// TIA Portal V15.1 export
// export: Created 2020-06-12T07:35:52.4755859Z, ExportSetting None, DisplayName Totally Integrated Automation Portal, DisplayVersion V15.1, DisplayName TIA Portal Openness, DisplayVersion V15.1, DisplayName STEP 7 Professional, DisplayVersion V15.1, DisplayName STEP 7 Safety, DisplayVersion V15.1, DisplayName WinCC Advanced, DisplayVersion V15.1
FUNCTION "MELT_Meas" : Void   // FC123, FBD
TITLE = Melt process measurements
{ S7_Optimized_Access := 'TRUE' }
// stored: SetENOAutomatically False
   VAR_TEMP
      trigger_ST : Bool;
      trigger_MT : Bool;
      trigger_HT : Bool;
      tTmpU : Real;
      tPower_set : Real;
      tReset_tara : Bool;
      tLimit : Bool;
      tAct_wt : Real;
      tWt_pres : Real;
      tWt_corr : Real;
      tWeight_av : Real;
      tMr_pres : Real;
      tPrs_corr : Real;
      tReset : Bool;
      tFactor : Real;
      tOperator_buttons_ok : Bool;
      tHt_ingot : Bool;
      tIngot_type : DInt;
      tConst_lim2_del_off : Bool;
      txxx : Bool;
      tSlag_molten : Bool;
      tClk_mr : Bool;
      tClk_sw : Bool;
      tCycle_mr : Time;
      tCycle_sw : Time;
      tWeight_av_1 : Real;
      tKWt : Real;
      par500 : Bool;
      par800 : Bool;
      par1050 : Bool;
      par1250 : Bool;
      tTot_ST : Real;
      tTot_time : Real;
      tTmp_time : Time;
      tT_ht : Time;
      tMeltrate1 : Real;
      tMeltrate2 : Real;
      tResMean : Real;
      tResStdDev : Real;
      tSync1 : Bool;
      tSync2 : Bool;
      tCTime1 : Time;
      tCTime2 : Time;
      tMRerr : Real;
      tSWerr : Real;
   END_VAR
BEGIN

REGION Network 1: Actual Power, kW
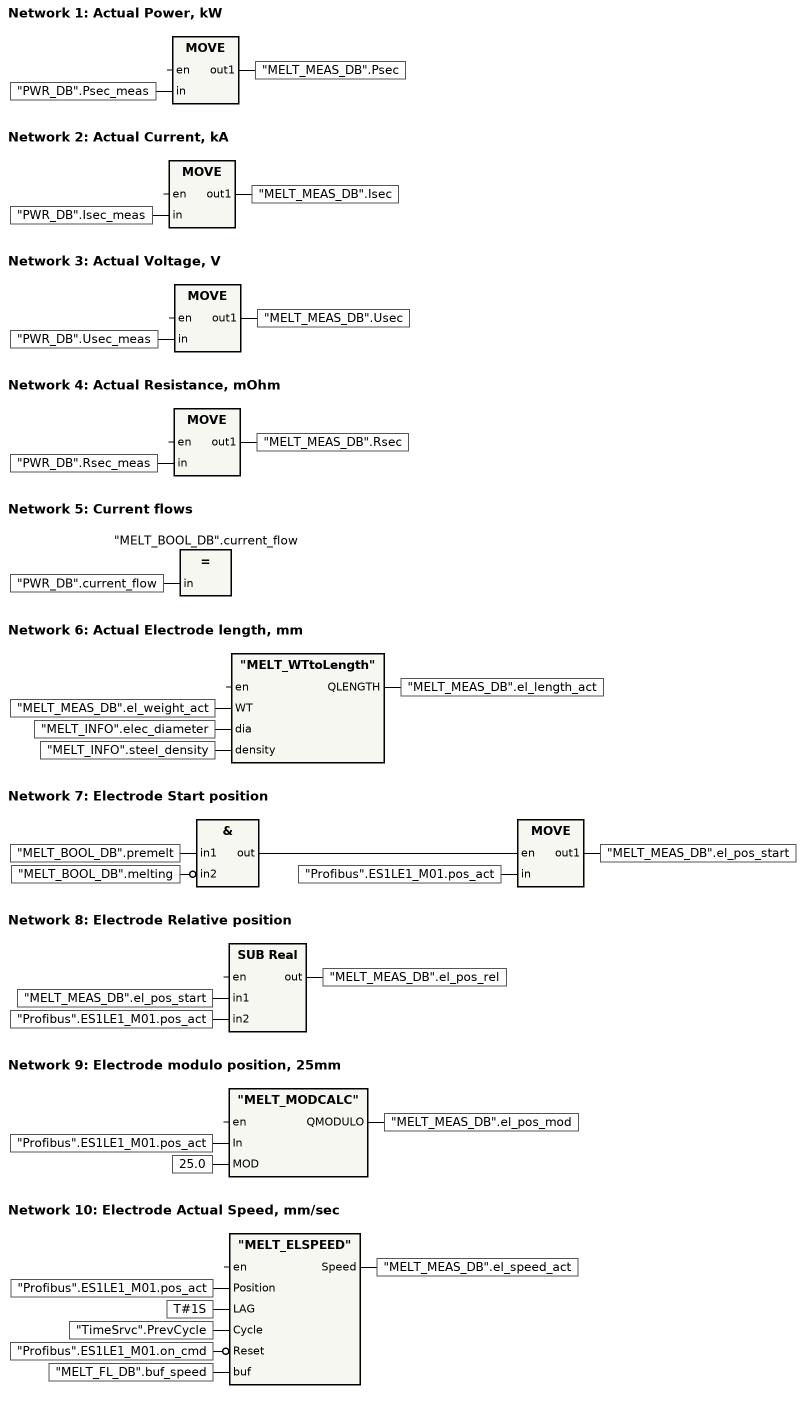
   "MELT_MEAS_DB".Psec := "PWR_DB".Psec_meas;
END_REGION

REGION Network 2: Actual Current, kA
   "MELT_MEAS_DB".Isec := "PWR_DB".Isec_meas;
END_REGION

REGION Network 3: Actual Voltage, V
   "MELT_MEAS_DB".Usec := "PWR_DB".Usec_meas;
END_REGION

REGION Network 4: Actual Resistance, mOhm
   "MELT_MEAS_DB".Rsec := "PWR_DB".Rsec_meas;
END_REGION

REGION Network 5: Current flows
   "MELT_BOOL_DB".current_flow := "PWR_DB".current_flow;
END_REGION

REGION Network 6: Actual Electrode length, mm
   "MELT_WTtoLength"(WT := "MELT_MEAS_DB".el_weight_act,
                     dia := "MELT_INFO".elec_diameter,
                     density := "MELT_INFO".steel_density,
                     QLENGTH => "MELT_MEAS_DB".el_length_act);
END_REGION

REGION Network 7: Electrode Start position
   IF "MELT_BOOL_DB".premelt AND NOT "MELT_BOOL_DB".melting THEN
       "MELT_MEAS_DB".el_pos_start := "Profibus".ES1LE1_M01.pos_act;
   END_IF;
END_REGION

REGION Network 8: Electrode Relative position
   "MELT_MEAS_DB".el_pos_rel := "MELT_MEAS_DB".el_pos_start - "Profibus".ES1LE1_M01.pos_act;
END_REGION

REGION Network 9: Electrode modulo position, 25mm
   "MELT_MODCALC"(In := "Profibus".ES1LE1_M01.pos_act, "MOD" := 25.0, QMODULO => "MELT_MEAS_DB".el_pos_mod);
END_REGION

REGION Network 10: Electrode Actual Speed, mm/sec
   "MELT_ELSPEED"(Position := "Profibus".ES1LE1_M01.pos_act,
                  LAG := T#1S,
                  Cycle := "TimeSrvc".PrevCycle,
                  Reset := NOT "Profibus".ES1LE1_M01.on_cmd,
                  buf := "MELT_FL_DB".buf_speed,
                  Speed => "MELT_MEAS_DB".el_speed_act);
END_REGION

REGION Network 11: Actual Ingot weight
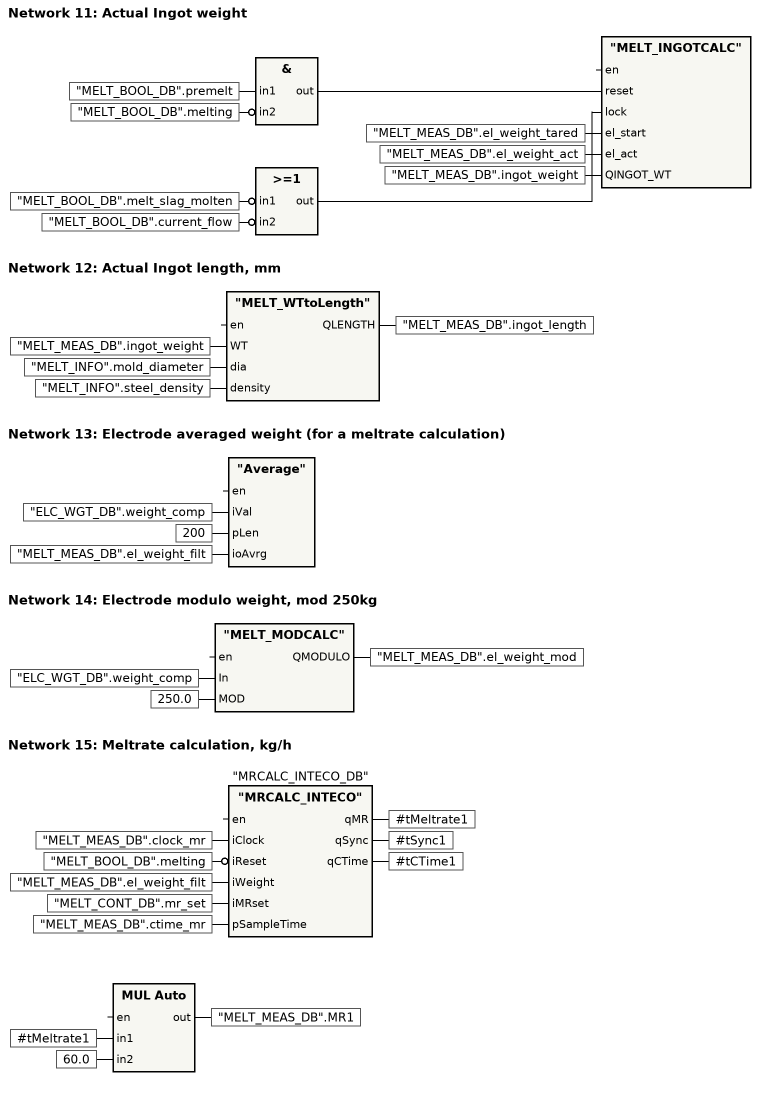
   "MELT_INGOTCALC"(reset := "MELT_BOOL_DB".premelt AND NOT "MELT_BOOL_DB".melting,
                    lock := NOT "MELT_BOOL_DB".melt_slag_molten OR NOT "MELT_BOOL_DB".current_flow,
                    el_start := "MELT_MEAS_DB".el_weight_tared,
                    el_act := "MELT_MEAS_DB".el_weight_act,
                    QINGOT_WT := "MELT_MEAS_DB".ingot_weight);
END_REGION

REGION Network 12: Actual Ingot length, mm
   "MELT_WTtoLength"(WT := "MELT_MEAS_DB".ingot_weight,
                     dia := "MELT_INFO".mold_diameter,
                     density := "MELT_INFO".steel_density,
                     QLENGTH => "MELT_MEAS_DB".ingot_length);
END_REGION

REGION Network 13: Electrode averaged weight (for a meltrate calculation)
   "Average"(iVal := "ELC_WGT_DB".weight_comp, pLen := 200, ioAvrg := "MELT_MEAS_DB".el_weight_filt);
END_REGION

REGION Network 14: Electrode modulo weight, mod 250kg
   "MELT_MODCALC"(In := "ELC_WGT_DB".weight_comp, "MOD" := 250.0, QMODULO => "MELT_MEAS_DB".el_weight_mod);
END_REGION

REGION Network 15: Meltrate calculation, kg/h
   "MRCALC_INTECO_DB"(iClock := "MELT_MEAS_DB".clock_mr,   // "MRCALC_INTECO"
                      iReset := NOT "MELT_BOOL_DB".melting,
                      iWeight := "MELT_MEAS_DB".el_weight_filt,
                      iMRset := "MELT_CONT_DB".mr_set,
                      pSampleTime := "MELT_MEAS_DB".ctime_mr,
                      qMR => #tMeltrate1,
                      qSync => #tSync1,
                      qCTime => #tCTime1);
   "MELT_MEAS_DB".MR1 := #tMeltrate1 * 60.0;
END_REGION

REGION Network 16: Meltrate calculation, kg/h (new)
   // from Boehler
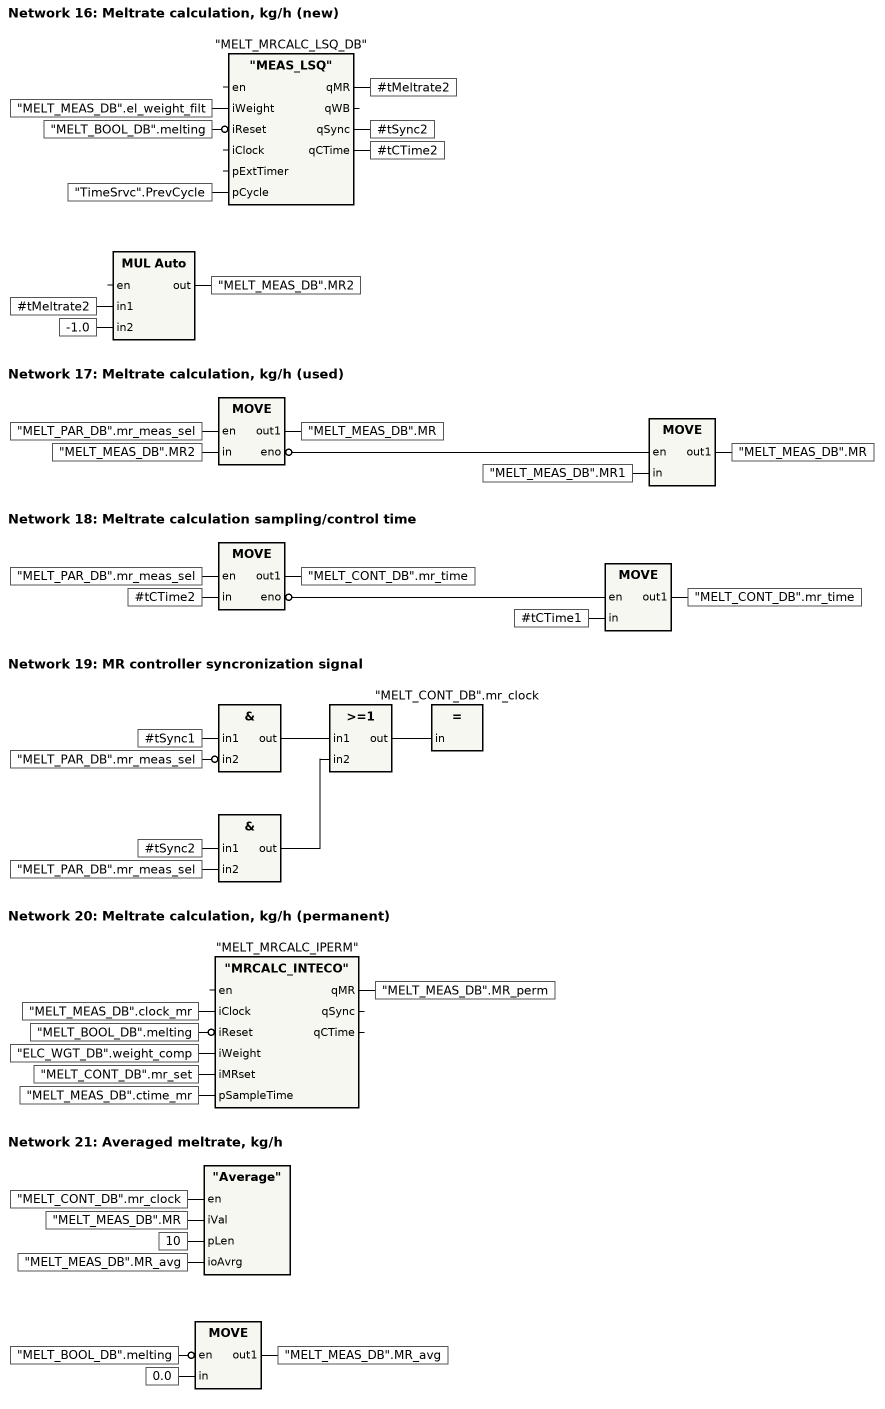
   "MELT_MRCALC_LSQ_DB"(iWeight := "MELT_MEAS_DB".el_weight_filt,   // "MEAS_LSQ"
                        iReset := NOT "MELT_BOOL_DB".melting,
                        pCycle := "TimeSrvc".PrevCycle,
                        qMR => #tMeltrate2,
                        qSync => #tSync2,
                        qCTime => #tCTime2);
   "MELT_MEAS_DB".MR2 := #tMeltrate2 * (-1.0);
END_REGION

REGION Network 17: Meltrate calculation, kg/h (used)
   IF "MELT_PAR_DB".mr_meas_sel THEN "MELT_MEAS_DB".MR := "MELT_MEAS_DB".MR2; END_IF;
   IF NOT "MELT_PAR_DB".mr_meas_sel THEN "MELT_MEAS_DB".MR := "MELT_MEAS_DB".MR1; END_IF;
END_REGION

REGION Network 18: Meltrate calculation sampling/control time
   IF "MELT_PAR_DB".mr_meas_sel THEN "MELT_CONT_DB".mr_time := #tCTime2; END_IF;
   IF NOT "MELT_PAR_DB".mr_meas_sel THEN "MELT_CONT_DB".mr_time := #tCTime1; END_IF;
END_REGION

REGION Network 19: MR controller syncronization signal
   "MELT_CONT_DB".mr_clock := (#tSync1 AND NOT "MELT_PAR_DB".mr_meas_sel) OR (#tSync2 AND "MELT_PAR_DB".mr_meas_sel);
END_REGION

REGION Network 20: Meltrate calculation, kg/h (permanent)
   "MELT_MRCALC_IPERM"(iClock := "MELT_MEAS_DB".clock_mr,   // "MRCALC_INTECO"
                       iReset := NOT "MELT_BOOL_DB".melting,
                       iWeight := "ELC_WGT_DB".weight_comp,
                       iMRset := "MELT_CONT_DB".mr_set,
                       pSampleTime := "MELT_MEAS_DB".ctime_mr,
                       qMR => "MELT_MEAS_DB".MR_perm);
END_REGION

REGION Network 21: Averaged meltrate, kg/h
   IF "MELT_CONT_DB".mr_clock THEN
       "Average"(iVal := "MELT_MEAS_DB".MR, pLen := 10, ioAvrg := "MELT_MEAS_DB".MR_avg);
   END_IF;
   IF NOT "MELT_BOOL_DB".melting THEN "MELT_MEAS_DB".MR_avg := 0.0; END_IF;
END_REGION

REGION Network 22: Swing calculation, mOhm
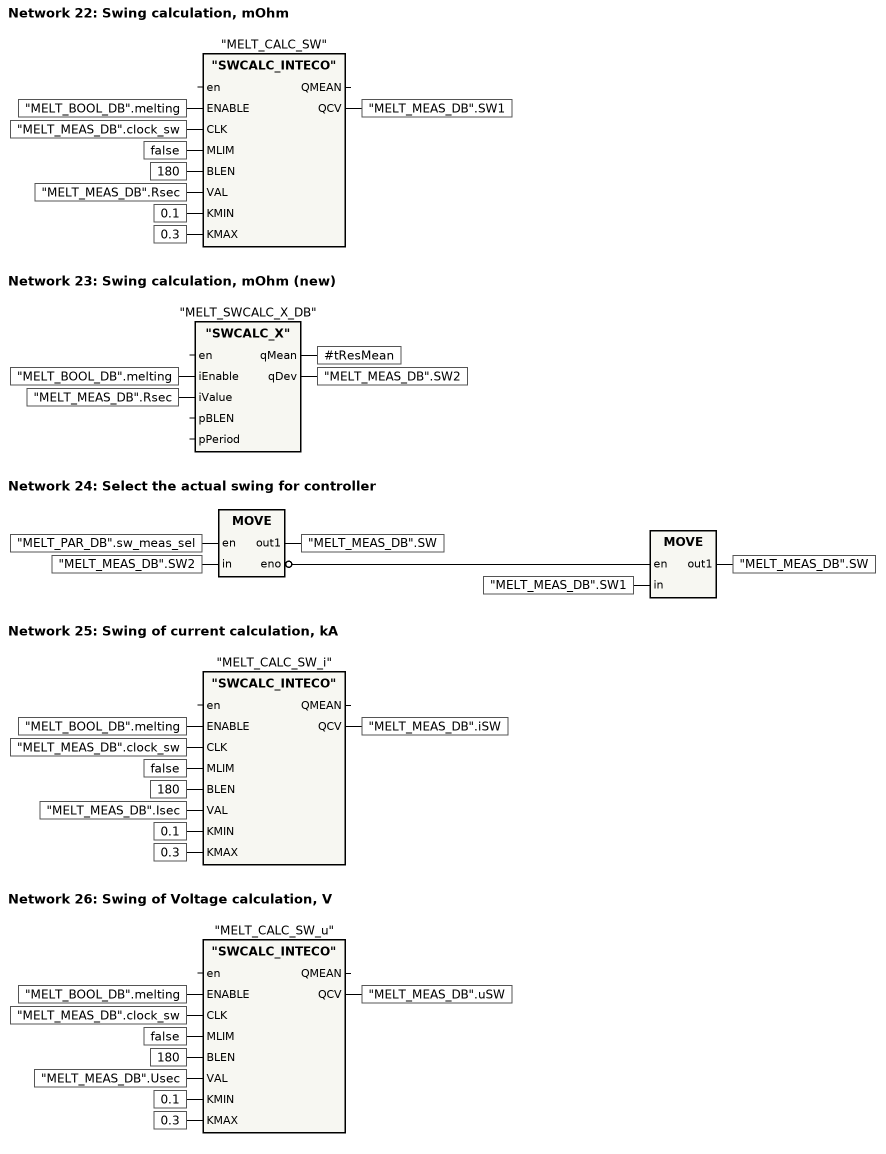
   "MELT_CALC_SW"(ENABLE := "MELT_BOOL_DB".melting,   // "SWCALC_INTECO"
                  CLK := "MELT_MEAS_DB".clock_sw,
                  MLIM := false,
                  BLEN := 180,
                  VAL := "MELT_MEAS_DB".Rsec,
                  KMIN := 0.1,
                  KMAX := 0.3,
                  QCV => "MELT_MEAS_DB".SW1);
END_REGION

REGION Network 23: Swing calculation, mOhm (new)
   // Mush better than old calculation
   "MELT_SWCALC_X_DB"(iEnable := "MELT_BOOL_DB".melting,   // "SWCALC_X"
                      iValue := "MELT_MEAS_DB".Rsec,
                      qMean => #tResMean,
                      qDev => "MELT_MEAS_DB".SW2);
END_REGION

REGION Network 24: Select the actual swing for controller
   IF "MELT_PAR_DB".sw_meas_sel THEN "MELT_MEAS_DB".SW := "MELT_MEAS_DB".SW2; END_IF;
   IF NOT "MELT_PAR_DB".sw_meas_sel THEN "MELT_MEAS_DB".SW := "MELT_MEAS_DB".SW1; END_IF;
END_REGION

REGION Network 25: Swing of current calculation, kA
   "MELT_CALC_SW_i"(ENABLE := "MELT_BOOL_DB".melting,   // "SWCALC_INTECO"
                    CLK := "MELT_MEAS_DB".clock_sw,
                    MLIM := false,
                    BLEN := 180,
                    VAL := "MELT_MEAS_DB".Isec,
                    KMIN := 0.1,
                    KMAX := 0.3,
                    QCV => "MELT_MEAS_DB".iSW);
END_REGION

REGION Network 26: Swing of Voltage calculation, V
   "MELT_CALC_SW_u"(ENABLE := "MELT_BOOL_DB".melting,   // "SWCALC_INTECO"
                    CLK := "MELT_MEAS_DB".clock_sw,
                    MLIM := false,
                    BLEN := 180,
                    VAL := "MELT_MEAS_DB".Usec,
                    KMIN := 0.1,
                    KMAX := 0.3,
                    QCV => "MELT_MEAS_DB".uSW);
END_REGION

REGION Network 27: Swing of Power calculation, kW
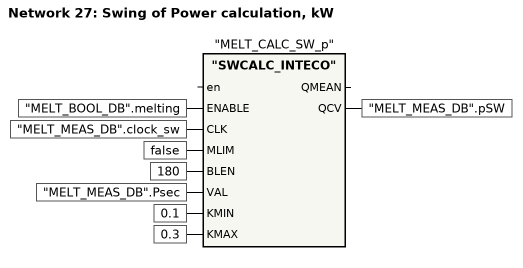
   "MELT_CALC_SW_p"(ENABLE := "MELT_BOOL_DB".melting,   // "SWCALC_INTECO"
                    CLK := "MELT_MEAS_DB".clock_sw,
                    MLIM := false,
                    BLEN := 180,
                    VAL := "MELT_MEAS_DB".Psec,
                    KMIN := 0.1,
                    KMAX := 0.3,
                    QCV => "MELT_MEAS_DB".pSW);
END_REGION

REGION Network 28: [Process error calculation]
END_REGION

REGION Network 29 (SCL): Meltrate error calculation
   IF ("MELT_CONT_DB".mr_set > 0)
       AND "MELT_BOOL_DB".melt_main_phase
       AND NOT "MELT_CONT_DB".mr_lock
   THEN
       #tMRerr := ABS(("MELT_CONT_DB".mr_act - "MELT_CONT_DB".mr_set) / "MELT_CONT_DB".mr_set);
   ELSE
       #tMRerr := 0.0;
   END_IF;
   "MELT_MEAS_DB".dMR := #tMRerr * 100.0;
END_REGION

REGION Network 30 (SCL): Swing error calculation
   IF "MELT_CONT_DB".sw_set > 0
       AND "MELT_BOOL_DB".melt_main_phase
       AND NOT "MELT_CONT_DB".sw_lock
   THEN
       #tSWerr := ABS(("MELT_CONT_DB".sw_act - "MELT_CONT_DB".sw_set) / "MELT_CONT_DB".sw_set);
   ELSE
       #tSWerr := 0.0;
   END_IF;
   "MELT_MEAS_DB".dSW := #tSWerr * 100.0;
END_REGION
END_FUNCTION
